// Library/Structures/AxesGroup/Acyclic/AxesGroupAcyclicAcrEntryRsp
{attribute 'pack_mode' := '1'} 
// ------------------------------------------------------------------------- 
//  SRCI Robot Library                                                
// ------------------------------------------------------------------------- 
//                                                                           
//  Object:      AxesGroupAcyclicAcrEntryRsp                                       
//  Author:      Thorsten Brach                                                
//  Date:        2024-06-01
//
//  Description:                                              
//   
//                                                                           
//  Copyright: 
//    (C) 2024 Thorsten Brach. All rights reserved                                                                                                                                            
//             Licensed under the LGPL-3.0 license.
//                                                                           
//  Disclaimer:                                                                           
//    This project is provided without any guarantee and can be used for   
//    private and commercial purposes. Any use is at the user’s 
//    own risk and responsibility.
//
// -------------------------------------------------------------------------
TYPE AxesGroupAcyclicAcrEntryRsp :
STRUCT
  /// Byte 00-03: Header
  Header : AxesGroupAcyclicAcrEntryRspHeader;
  /// Byte 04-07: Trigger sub header
  Trigger : AxesGroupAcyclicAcrEntryRspTrigger;
  /// Byte 08-xx: RSP Payload defined by type per CMD definition. Generated by Appl. Layer Task
  Payload : ARRAY[0..RobotLibraryParameter.TELEGRAM_PAYLOAD_MAX] OF BYTE;    
END_STRUCT
END_TYPE

// Library/Structures/AxesGroup/Acyclic/AxesGroupAcyclicAcrEntryRspBuffer
{attribute 'pack_mode' := '1'} 
// ------------------------------------------------------------------------- 
//  SRCI Robot Library                                                
// ------------------------------------------------------------------------- 
//                                                                           
//  Object:      AxesGroupAcyclicAcrEntryRspBuffer                                       
//  Author:      Thorsten Brach                                                
//  Date:        2024-06-01
//
//  Description:                                              
//   
//                                                                           
//  Copyright: 
//    (C) 2024 Thorsten Brach. All rights reserved                                                                                                                                            
//             Licensed under the LGPL-3.0 license.
//                                                                           
//  Disclaimer:                                                                           
//    This project is provided without any guarantee and can be used for   
//    private and commercial purposes. Any use is at the user’s 
//    own risk and responsibility.
//
// -------------------------------------------------------------------------
TYPE AxesGroupAcyclicAcrEntryRspBuffer :
STRUCT
  /// Timestamp
  Timestamp         : SystemTime;
  ///
  State             : BufferStateRsp;
  /// Payload defined by type per CMD definition. Processed by Appl. Layer Task.
  Payload           : ARRAY[0..RobotLibraryParameter.TELEGRAM_PAYLOAD_MAX] OF BYTE;
  /// Payload length
  PayloadLen        : UDINT;  
  /// Payload poiner   
  PayLoadPtr        : DWORD;
END_STRUCT
END_TYPE

// Library/Structures/AxesGroup/Acyclic/AxesGroupAcyclicAcrEntryRspHeader
{attribute 'pack_mode' := '1'} 
// ------------------------------------------------------------------------- 
//  SRCI Robot Library                                                
// ------------------------------------------------------------------------- 
//                                                                           
//  Object:      AxesGroupAcyclicAcrEntryRspHeader                                       
//  Author:      Thorsten Brach                                                
//  Date:        2024-06-01
//
//  Description:                                              
//   
//                                                                           
//  Copyright: 
//    (C) 2024 Thorsten Brach. All rights reserved                                                                                                                                            
//             Licensed under the LGPL-3.0 license.
//                                                                           
//  Disclaimer:                                                                           
//    This project is provided without any guarantee and can be used for   
//    private and commercial purposes. Any use is at the user’s 
//    own risk and responsibility.
//
// -------------------------------------------------------------------------
TYPE AxesGroupAcyclicAcrEntryRspHeader :
STRUCT
  /// Byte 00 : State  (Bit 0..3)
  State                : CmdMessageState; // ToDo : nicht sicher ob das richtig ist 
  /// Byte 00 : ParSeq (Bit 4..5)
  ParSeq               : BYTE;
  /// Byte 01 : Alarm Message Severity
  AlarmMessageSeverity : Severity;
  /// Byte 02 : Alarm Message Code
  AlarmMessageCode     : UINT;  
END_STRUCT
END_TYPE

// Library/Structures/AxesGroup/Acyclic/AxesGroupAcyclicAcrEntryRspTrigger
{attribute 'pack_mode' := '1'} 
// ------------------------------------------------------------------------- 
//  SRCI Robot Library                                                
// ------------------------------------------------------------------------- 
//                                                                           
//  Object:      AxesGroupAcyclicAcrEntryRspTrigger                                       
//  Author:      Thorsten Brach                                                
//  Date:        2024-06-01
//
//  Description:                                              
//   
//                                                                           
//  Copyright: 
//    (C) 2024 Thorsten Brach. All rights reserved                                                                                                                                            
//             Licensed under the LGPL-3.0 license.
//                                                                           
//  Disclaimer:                                                                           
//    This project is provided without any guarantee and can be used for   
//    private and commercial purposes. Any use is at the user’s 
//    own risk and responsibility.
//
// -------------------------------------------------------------------------
TYPE AxesGroupAcyclicAcrEntryRspTrigger :
STRUCT
  /// Number of Trigger based CMD invocations
  InvocationCounter       : USINT;
  /// Number of missed Triggers
  MissedInvocationCounter : USINT;
  /// FollowID of Trigger initiator
  OriginID                : WORD;
END_STRUCT
END_TYPE

// Library/Structures/AxesGroup/Acyclic/AxesGroupAcyclicExecutionOrderList
{attribute 'pack_mode' := '1'} 
// ------------------------------------------------------------------------- 
//  SRCI Robot Library                                                
// ------------------------------------------------------------------------- 
//                                                                           
//  Object:      AxesGroupAcyclicExecutionOrderList                                       
//  Author:      Thorsten Brach                                                
//  Date:        2024-06-01
//
//  Description:                                              
//   
//                                                                           
//  Copyright: 
//    (C) 2024 Thorsten Brach. All rights reserved                                                                                                                                            
//             Licensed under the LGPL-3.0 license.
//                                                                           
//  Disclaimer:                                                                           
//    This project is provided without any guarantee and can be used for   
//    private and commercial purposes. Any use is at the user’s 
//    own risk and responsibility.
//
// -------------------------------------------------------------------------
TYPE AxesGroupAcyclicExecutionOrderList :
STRUCT
  /// Command
  Command  : ARRAY [1..RobotLibraryParameter.ACTIVE_CMD_REGISTER_ENTRIES_MAX] OF UINT;
  /// Response
  Response : ARRAY [1..RobotLibraryParameter.ACTIVE_CMD_REGISTER_ENTRIES_MAX] OF UINT;
END_STRUCT
END_TYPE

// Library/Structures/AxesGroup/Cyclic/AxesGroupCyclic
{attribute 'pack_mode' := '1'} 
// ------------------------------------------------------------------------- 
//  SRCI Robot Library                                                
// ------------------------------------------------------------------------- 
//                                                                           
//  Object:      AxesGroupCyclic                                       
//  Author:      Thorsten Brach                                                
//  Date:        2024-06-01
//
//  Description:                                              
//   
//                                                                           
//  Copyright: 
//    (C) 2024 Thorsten Brach. All rights reserved                                                                                                                                            
//             Licensed under the LGPL-3.0 license.
//                                                                           
//  Disclaimer:                                                                           
//    This project is provided without any guarantee and can be used for   
//    private and commercial purposes. Any use is at the user’s 
//    own risk and responsibility.
//
// -------------------------------------------------------------------------
TYPE AxesGroupCyclic :
STRUCT
  /// Cyclic data from PLC to Robot 
  PlcToRob : AxesGroupCyclicPlcToRob;
  /// Cyclic data from Robot to PLC
  RobToPlc : AxesGroupCyclicRobToPlc;
END_STRUCT
END_TYPE

// Library/Structures/AxesGroup/Cyclic/AxesGroupCyclicPlcToRob
{attribute 'pack_mode' := '1'} 
// ------------------------------------------------------------------------- 
//  SRCI Robot Library                                                
// ------------------------------------------------------------------------- 
//                                                                           
//  Object:      AxesGroupCyclicPlcToRob                                       
//  Author:      Thorsten Brach                                                
//  Date:        2024-06-01
//
//  Description:                                              
//   
//                                                                           
//  Copyright: 
//    (C) 2024 Thorsten Brach. All rights reserved                                                                                                                                            
//             Licensed under the LGPL-3.0 license.
//                                                                           
//  Disclaimer:                                                                           
//    This project is provided without any guarantee and can be used for   
//    private and commercial purposes. Any use is at the user’s 
//    own risk and responsibility.
//
// -------------------------------------------------------------------------
TYPE AxesGroupCyclicPlcToRob :
STRUCT
  /// Version of SRCI specification
  /// Bit 0-4 : Minor version = Features        (0..31)
  /// Bit 5-7 : Major version = Breaking change (0..07)
  SRCIVersion            : VersionStruct;
  /// Fast stop trigger 
  FastStop               : BYTE;
  /// Connection alive signal
  LifeSign               : BYTE;
  /// Number of Bytes of the frame to be used for the telegram of the given Axisgroup. Direction client to server
  TelegramLengthPlcToRob : UINT;
  /// Number of Bytes of the frame to be used for the telegram of the given Axisgroup. Direction server to client
  TelegramLengthRobToPlc : UINT;
  /// Control AxesGroupID Telegtam state control
  AxesGroupID            : BYTE;
  /// Telegram state control
  Control                : ControlHalfByte;
  /// Reserved for later versions
  Reserved               : BYTE;
  /// Configuration of the optional cyclic data. Direction client to server
  TelegramNumberPlcToRob : UINT;
  /// Configuration of the optional cyclic data. Direction server to client
  TelegramNumberRobToPlc : UINT;
  /// Date of the client in the format days since 1990.01.01
  ClientDate             : IEC_DATE;
  /// Time in the clients time zone in the format milliseconds since start of day
  ClientTime             : IEC_TIME;    
  ///Index of tool of returned position
  /// •     -1: Currently used tool on RC
  /// •      0: Flange (default)
  /// • 1..254: Tool frames
  ToolNo                 : INT;
  /// Index of frame of returned position
  /// •     -1: Currently used frame on RC
  /// •      0: WCS (default)
  /// • 1..254: User frames
  FrameNo                : INT;
END_STRUCT
END_TYPE

// Library/Structures/AxesGroup/Cyclic/AxesGroupCyclicRobToPlc
{attribute 'pack_mode' := '1'} 
// ------------------------------------------------------------------------- 
//  SRCI Robot Library                                                
// ------------------------------------------------------------------------- 
//                                                                           
//  Object:      AxesGroupCyclicRobToPlc                                       
//  Author:      Thorsten Brach                                                
//  Date:        2024-06-01
//
//  Description:                                              
//   
//                                                                           
//  Copyright: 
//    (C) 2024 Thorsten Brach. All rights reserved                                                                                                                                            
//             Licensed under the LGPL-3.0 license.
//                                                                           
//  Disclaimer:                                                                           
//    This project is provided without any guarantee and can be used for   
//    private and commercial purposes. Any use is at the user’s 
//    own risk and responsibility.
//
// -------------------------------------------------------------------------
TYPE AxesGroupCyclicRobToPlc :
STRUCT
  /// Version of SRCI specification
  /// Bit 0-4 : Minor version = Features        (0..31)
  /// Bit 5-7 : Major version = Breaking change (0..07)
  SRCIVersion   : VersionStruct;
  /// Connection alive signal
  LifeSign      : BYTE;
  /// Reserved byte
  Reserved      : BYTE;
  /// Initialization and Telegram control state
  TelegramState : TelegramState;
  /// Combination of various RA related states.
  StatusRobotArm: RaStatusWord;
  /// Actual override in percentage encoding 
  Override      : UINT;  
END_STRUCT
END_TYPE

// Library/Structures/AxesGroup/CyclicOptional/Internal/AxesGroupCyclicOptionalDataCartesianPosition
{attribute 'pack_mode' := '1'} 
// ------------------------------------------------------------------------- 
//  SRCI Robot Library                                                
// ------------------------------------------------------------------------- 
//                                                                           
//  Object:      AxesGroupCyclicOptionalDataCartesianPosition                                       
//  Author:      Thorsten Brach                                                
//  Date:        2024-06-01
//
//  Description:                                              
//   
//                                                                           
//  Copyright: 
//    (C) 2024 Thorsten Brach. All rights reserved                                                                                                                                            
//             Licensed under the LGPL-3.0 license.
//                                                                           
//  Disclaimer:                                                                           
//    This project is provided without any guarantee and can be used for   
//    private and commercial purposes. Any use is at the user’s 
//    own risk and responsibility.
//
// -------------------------------------------------------------------------
TYPE AxesGroupCyclicOptionalDataCartesianPosition EXTENDS  RobotCartesianPositionShort :
STRUCT
  /// indicates that this optional parameter will be used
  Active           : BOOL;
  /// corresponding coordinate systems
  CoordinateSystem : RobotCoordinateSystemParameters; 
END_STRUCT
END_TYPE

// Library/Structures/AxesGroup/CyclicOptional/Internal/AxesGroupCyclicOptionalDataCartesianPositionExt
{attribute 'pack_mode' := '1'} 
// ------------------------------------------------------------------------- 
//  SRCI Robot Library                                                
// ------------------------------------------------------------------------- 
//                                                                           
//  Object:      AxesGroupCyclicOptionalDataCartesianPositionExt                                       
//  Author:      Thorsten Brach                                                
//  Date:        2024-06-01
//
//  Description:                                              
//   
//                                                                           
//  Copyright: 
//    (C) 2024 Thorsten Brach. All rights reserved                                                                                                                                            
//             Licensed under the LGPL-3.0 license.
//                                                                           
//  Disclaimer:                                                                           
//    This project is provided without any guarantee and can be used for   
//    private and commercial purposes. Any use is at the user’s 
//    own risk and responsibility.
//
// -------------------------------------------------------------------------
TYPE AxesGroupCyclicOptionalDataCartesianPositionExt EXTENDS RobotCartesianPositionExt :
STRUCT
  /// indicates that this optional parameter will be used
  Active : BOOL;
END_STRUCT
END_TYPE

// Library/Structures/AxesGroup/CyclicOptional/Internal/AxesGroupCyclicOptionalDataCurrent
{attribute 'pack_mode' := '1'} 
// ------------------------------------------------------------------------- 
//  SRCI Robot Library                                                
// ------------------------------------------------------------------------- 
//                                                                           
//  Object:      AxesGroupCyclicOptionalDataJointCurrent                                       
//  Author:      Thorsten Brach                                                
//  Date:        2024-06-01
//
//  Description:                                              
//   
//                                                                           
//  Copyright: 
//    (C) 2024 Thorsten Brach. All rights reserved                                                                                                                                            
//             Licensed under the LGPL-3.0 license.
//                                                                           
//  Disclaimer:                                                                           
//    This project is provided without any guarantee and can be used for   
//    private and commercial purposes. Any use is at the user’s 
//    own risk and responsibility.
//
// -------------------------------------------------------------------------
TYPE AxesGroupCyclicOptionalDataCurrent EXTENDS RobotJointCurrentShort :
STRUCT
    /// indicates that this optional parameter will be used
  Active : BOOL;
END_STRUCT
END_TYPE

// Library/Structures/AxesGroup/CyclicOptional/Internal/AxesGroupCyclicOptionalDataCurrentExt
{attribute 'pack_mode' := '1'} 
// ------------------------------------------------------------------------- 
//  SRCI Robot Library                                                
// ------------------------------------------------------------------------- 
//                                                                           
//  Object:      AxesGroupCyclicOptionalDataJointCurrentExt                                       
//  Author:      Thorsten Brach                                                
//  Date:        2024-06-01
//
//  Description:                                              
//   
//                                                                           
//  Copyright: 
//    (C) 2024 Thorsten Brach. All rights reserved                                                                                                                                            
//             Licensed under the LGPL-3.0 license.
//                                                                           
//  Disclaimer:                                                                           
//    This project is provided without any guarantee and can be used for   
//    private and commercial purposes. Any use is at the user’s 
//    own risk and responsibility.
//
// -------------------------------------------------------------------------
TYPE AxesGroupCyclicOptionalDataCurrentExt EXTENDS RobotJointCurrentExt :
STRUCT
    /// indicates that this optional parameter will be used
  Active : BOOL;
END_STRUCT
END_TYPE

// Library/Structures/AxesGroup/CyclicOptional/Internal/AxesGroupCyclicOptionalDataForce
{attribute 'pack_mode' := '1'} 
// ------------------------------------------------------------------------- 
//  SRCI Robot Library                                                
// ------------------------------------------------------------------------- 
//                                                                           
//  Object:      AxesGroupCyclicOptionalDataCartesianForce                                       
//  Author:      Thorsten Brach                                                
//  Date:        2024-06-01
//
//  Description:                                              
//   
//                                                                           
//  Copyright: 
//    (C) 2024 Thorsten Brach. All rights reserved                                                                                                                                            
//             Licensed under the LGPL-3.0 license.
//                                                                           
//  Disclaimer:                                                                           
//    This project is provided without any guarantee and can be used for   
//    private and commercial purposes. Any use is at the user’s 
//    own risk and responsibility.
//
// -------------------------------------------------------------------------
TYPE AxesGroupCyclicOptionalDataForce EXTENDS RobotCartesianForceShort:
STRUCT
  /// indicates that this optional parameter will be used
  Active           : BOOL;
END_STRUCT
END_TYPE

// Library/Structures/AxesGroup/CyclicOptional/Internal/AxesGroupCyclicOptionalDataForceExt
{attribute 'pack_mode' := '1'} 
// ------------------------------------------------------------------------- 
//  SRCI Robot Library                                                
// ------------------------------------------------------------------------- 
//                                                                           
//  Object:      AxesGroupCyclicOptionalDataCartesianForceExt                                       
//  Author:      Thorsten Brach                                                
//  Date:        2024-06-01
//
//  Description:                                              
//   
//                                                                           
//  Copyright: 
//    (C) 2024 Thorsten Brach. All rights reserved                                                                                                                                            
//             Licensed under the LGPL-3.0 license.
//                                                                           
//  Disclaimer:                                                                           
//    This project is provided without any guarantee and can be used for   
//    private and commercial purposes. Any use is at the user’s 
//    own risk and responsibility.
//
// -------------------------------------------------------------------------
TYPE AxesGroupCyclicOptionalDataForceExt EXTENDS RobotCartesianForceExt:
STRUCT
  /// indicates that this optional parameter will be used
  Active           : BOOL;
END_STRUCT
END_TYPE

// Library/Structures/AxesGroup/CyclicOptional/Internal/AxesGroupCyclicOptionalDataJointPosition
{attribute 'pack_mode' := '1'} 
// ------------------------------------------------------------------------- 
//  SRCI Robot Library                                                
// ------------------------------------------------------------------------- 
//                                                                           
//  Object:      AxesGroupCyclicOptionalDataJointPosition                                       
//  Author:      Thorsten Brach                                                
//  Date:        2024-06-01
//
//  Description:                                              
//   
//                                                                           
//  Copyright: 
//    (C) 2024 Thorsten Brach. All rights reserved                                                                                                                                            
//             Licensed under the LGPL-3.0 license.
//                                                                           
//  Disclaimer:                                                                           
//    This project is provided without any guarantee and can be used for   
//    private and commercial purposes. Any use is at the user’s 
//    own risk and responsibility.
//
// -------------------------------------------------------------------------
TYPE AxesGroupCyclicOptionalDataJointPosition EXTENDS RobotJointPositionShort :
STRUCT
    /// indicates that this optional parameter will be used
  Active : BOOL;
END_STRUCT
END_TYPE

// Library/Structures/AxesGroup/CyclicOptional/Internal/AxesGroupCyclicOptionalDataJointPositionExt
{attribute 'pack_mode' := '1'} 
// ------------------------------------------------------------------------- 
//  SRCI Robot Library                                                
// ------------------------------------------------------------------------- 
//                                                                           
//  Object:      AxesGroupCyclicOptionalDataJointPositionExt                                       
//  Author:      Thorsten Brach                                                
//  Date:        2024-06-01
//
//  Description:                                              
//   
//                                                                           
//  Copyright: 
//    (C) 2024 Thorsten Brach. All rights reserved                                                                                                                                            
//             Licensed under the LGPL-3.0 license.
//                                                                           
//  Disclaimer:                                                                           
//    This project is provided without any guarantee and can be used for   
//    private and commercial purposes. Any use is at the user’s 
//    own risk and responsibility.
//
// -------------------------------------------------------------------------
TYPE AxesGroupCyclicOptionalDataJointPositionExt EXTENDS RobotJointPositionExt :
STRUCT
    /// indicates that this optional parameter will be used
  Active : BOOL;
END_STRUCT
END_TYPE

// Library/Structures/AxesGroup/CyclicOptional/Internal/AxesGroupCyclicOptionalDataSubProgram
{attribute 'pack_mode' := '1'} 
// ------------------------------------------------------------------------- 
//  SRCI Robot Library                                                
// ------------------------------------------------------------------------- 
//                                                                           
//  Object:      AxesGroupCyclicOptionalDataSubProgram                                       
//  Author:      Thorsten Brach                                                
//  Date:        2024-06-01
//
//  Description:                                              
//   
//                                                                           
//  Copyright: 
//    (C) 2024 Thorsten Brach. All rights reserved                                                                                                                                            
//             Licensed under the LGPL-3.0 license.
//                                                                           
//  Disclaimer:                                                                           
//    This project is provided without any guarantee and can be used for   
//    private and commercial purposes. Any use is at the user’s 
//    own risk and responsibility.
//
// -------------------------------------------------------------------------
TYPE AxesGroupCyclicOptionalDataSubProgram EXTENDS RobotSubProgramData :
STRUCT
  /// indicates that this optional parameter will be used
  Active : BOOL;
END_STRUCT
END_TYPE

// Library/Structures/AxesGroup/CyclicOptional/AxesGroupCyclicOptionalData
{attribute 'pack_mode' := '1'} 
// ------------------------------------------------------------------------- 
//  SRCI Robot Library                                                
// ------------------------------------------------------------------------- 
//                                                                           
//  Object:      AxesGroupCyclicOptionalData                                       
//  Author:      Thorsten Brach                                                
//  Date:        2024-06-01
//
//  Description:                                              
//   
//                                                                           
//  Copyright: 
//    (C) 2024 Thorsten Brach. All rights reserved                                                                                                                                            
//             Licensed under the LGPL-3.0 license.
//                                                                           
//  Disclaimer:                                                                           
//    This project is provided without any guarantee and can be used for   
//    private and commercial purposes. Any use is at the user’s 
//    own risk and responsibility.
//
// -------------------------------------------------------------------------
TYPE AxesGroupCyclicOptionalData :
STRUCT
  /// Optional cyclic data from PLC to Robot
  PlcToRob : AxesGroupCyclicOptionalDataPlcToRob;
  /// Optional cyclic data from Robot to PLC
  RobToPlc : AxesGroupCyclicOptionalDataRobToPlc;
END_STRUCT
END_TYPE

// Library/Structures/AxesGroup/CyclicOptional/AxesGroupCyclicOptionalDataPlcToRob
{attribute 'pack_mode' := '1'} 
// ------------------------------------------------------------------------- 
//  SRCI Robot Library                                                
// ------------------------------------------------------------------------- 
//                                                                           
//  Object:      vAxesGroupCyclicOptionalDataPlcToRob                                       
//  Author:      Thorsten Brach                                                
//  Date:        2024-06-01
//
//  Description:                                              
//   
//                                                                           
//  Copyright: 
//    (C) 2024 Thorsten Brach. All rights reserved                                                                                                                                            
//             Licensed under the LGPL-3.0 license.
//                                                                           
//  Disclaimer:                                                                           
//    This project is provided without any guarantee and can be used for   
//    private and commercial purposes. Any use is at the user’s 
//    own risk and responsibility.
//
// -------------------------------------------------------------------------
TYPE AxesGroupCyclicOptionalDataPlcToRob :
STRUCT
  /// Transmit cyclic data from PLC to RC for the usage in a subprogram on the RC called via the function “CallSubprogram”
  SubProgramData        :  AxesGroupCyclicOptionalDataSubProgram;
  /// short cartesian position with TCP position (X, Y,Z), rotation (RX, RY, RZ), configuration bytes (Config, TurnNumber), position of first external axis (E1) and corresponding coordinate systems (ToolNo, FrameNo)
  CartesianPosition     :  AxesGroupCyclicOptionalDataCartesianPosition;
  /// the external axis values for an extended cartesian position (E2, E3, E4, E5, E6) 
  /// When selected, Tool and Frame will automatically cyclically be sent from client to server.
  CartesianPositionExt  :  AxesGroupCyclicOptionalDataCartesianPositionExt;
  /// short axes position with joint values (J1, J2, J3,J4, J5, J6) and position of first external axis (E1)
  JointPosition         :  AxesGroupCyclicOptionalDataJointPosition;
  /// the external axis values for an extended joint position (E2, E3, E4, E5, E6)
  JointPositionExt      :  AxesGroupCyclicOptionalDataJointPositionExt;
  /// force with the divided forces in the individual directions (X, Y, Z, RX, RY, RZ)
  Force                 :  AxesGroupCyclicOptionalDataForce;
  /// current force for the external axis (E1, E2, E3, E4, E5, E6)
  ForceExt              :  AxesGroupCyclicOptionalDataForceExt;
END_STRUCT
END_TYPE

// Library/Structures/AxesGroup/CyclicOptional/AxesGroupCyclicOptionalDataRobToPlc
{attribute 'pack_mode' := '1'} 
// ------------------------------------------------------------------------- 
//  SRCI Robot Library                                                
// ------------------------------------------------------------------------- 
//                                                                           
//  Object:      AxesGroupCyclicOptionalDataRobToPlc                                       
//  Author:      Thorsten Brach                                                
//  Date:        2024-06-01
//
//  Description:                                              
//   
//                                                                           
//  Copyright: 
//    (C) 2024 Thorsten Brach. All rights reserved                                                                                                                                            
//             Licensed under the LGPL-3.0 license.
//                                                                           
//  Disclaimer:                                                                           
//    This project is provided without any guarantee and can be used for   
//    private and commercial purposes. Any use is at the user’s 
//    own risk and responsibility.
//
// -------------------------------------------------------------------------
TYPE AxesGroupCyclicOptionalDataRobToPlc :
STRUCT
  /// Transmit cyclic data from PLC to RC for the usage in a subprogram on the RC called via the function “CallSubprogram”
  SubProgramData        :  AxesGroupCyclicOptionalDataSubProgram;
  /// short cartesian position with TCP position (X, Y,Z), rotation (RX, RY, RZ), configuration bytes (Config, TurnNumber), position of first external axis (E1) and corresponding coordinate systems (ToolNo, FrameNo)
  CartesianPosition     :  AxesGroupCyclicOptionalDataCartesianPosition;
  /// the external axis values for an extended cartesian position (E2, E3, E4, E5, E6) 
  /// When selected, Tool and Frame will automatically cyclically be sent from client to server.
  CartesianPositionExt  :  AxesGroupCyclicOptionalDataCartesianPositionExt;
  /// short axes position with joint values (J1, J2, J3,J4, J5, J6) and position of first external axis (E1)
  JointPosition         :  AxesGroupCyclicOptionalDataJointPosition;
  /// the external axis values for an extended joint position (E2, E3, E4, E5, E6)
  JointPositionExt      :  AxesGroupCyclicOptionalDataJointPositionExt;
  /// force with the divided forces in the individual directions (X, Y, Z, RX, RY, RZ)
  Force                 :  AxesGroupCyclicOptionalDataForce;
  /// current force for the external axis (E1, E2, E3, E4, E5, E6)
  ForceExt              :  AxesGroupCyclicOptionalDataForceExt;
  /// ctual axes current of individual axes (J1, J2, J3, J4, J5, J6)
  Current               :  AxesGroupCyclicOptionalDataCurrent;
  /// actual current for the external axis (E1, E2,E3, E4, E5, E6)
  CurrentExt            :  AxesGroupCyclicOptionalDataCurrentExt;  
END_STRUCT
END_TYPE

// Library/Structures/AxesGroup/InternalData/AxesGroupInternalData
{attribute 'pack_mode' := '1'} 
// ------------------------------------------------------------------------- 
//  SRCI Robot Library                                                
// ------------------------------------------------------------------------- 
//                                                                           
//  Object:      AxesGroup                                       
//  Author:      Thorsten Brach                                                
//  Date:        2024-08-28
//
//  Description:                                              
//   
//                                                                           
//  Copyright: 
//    (C) 2024 Thorsten Brach. All rights reserved                                                                                                                                            
//             Licensed under the LGPL-3.0 license.
//                                                                           
//  Disclaimer:                                                                           
//    This project is provided without any guarantee and can be used for   
//    private and commercial purposes. Any use is at the user’s 
//    own risk and responsibility.
//
// -------------------------------------------------------------------------
TYPE AxesGroupInternalData :
STRUCT
  /// Current System Time
  SystemTime           : SystemTime;
    /// • TRUE: Function is supported by RC • FALSE: Function is not supported by RC See Table 6-14 for bit assignment.
  RCSupportedFunctions : RCSupportedFunctions;
  /// Online Change detected
  OnlineChange         : BOOL;  
  /// Rising edge for Online Change detected
  OnlineChange_R       : R_TRIG;  
  /// Falling edge for Online Change detected
  OnlineChange_F       : F_TRIG;  
  /// GroupReset active
  GroupReset           : BOOL; 
  /// Rising edge for GroupReset
  GroupReset_R         : R_TRIG;  
  /// Falling edge for GroupReset
  GroupReset_F         : F_TRIG;
  /// Counter of sequences to send
  SequenceCountSend    : DINT;
  /// Counter of sequences received
  SequenceCountRecv    : DINT;
  /// Counter of fragments to send
  FragmentCountSend    : ARRAY[0..1] OF DINT;
  /// Counter of fragments received
  FragmentCountRecv    : ARRAY[0..1] OF DINT;
  /// Current Sequence ID
  CurrentSEQ           : ARRAY[0..1] OF UINT;
  /// Current acknowledge ID
  CurrentACK           : ARRAY[0..1] OF UINT;  
  /// Current Sequence ID has changed -> send new data 
  NewSEQ               : ARRAY[0..1] OF BOOL;
  /// Last received acknowledge ID
  LastACK              : ARRAY[0..1] OF UINT;  
END_STRUCT
END_TYPE

// Library/Structures/AxesGroup/MessageLog/AxesGroupMessageLog
{attribute 'pack_mode' := '1'} 
// ------------------------------------------------------------------------- 
//  SRCI Robot Library                                                
// ------------------------------------------------------------------------- 
//                                                                           
//  Object:      AxesGroupMessageLog                                       
//  Author:      Thorsten Brach                                                
//  Date:        2024-06-01
//
//  Description:                                              
//   
//                                                                           
//  Copyright: 
//    (C) 2024 Thorsten Brach. All rights reserved                                                                                                                                            
//             Licensed under the LGPL-3.0 license.
//                                                                           
//  Disclaimer:                                                                           
//    This project is provided without any guarantee and can be used for   
//    private and commercial purposes. Any use is at the user’s 
//    own risk and responsibility.
//
// -------------------------------------------------------------------------
TYPE AxesGroupMessageLog :
STRUCT
  /// Amount of system log entries
  SystemLogEntries : UINT := DINT_TO_UINT(RobotLibraryParameter.SYSTEM_LOG_MAX);
  /// Amount of message log entries
  MessagesEntries  : UINT := DINT_TO_UINT(RobotLibraryParameter.MESSAGE_LOG_MAX);
  /// Logging level
  LogLevel         : LogLevel;
  /// System log
  SystemLog        : ARRAY[0..RobotLibraryParameter.SYSTEM_LOG_MAX] OF STRING(255);
  /// Message Log
  Messages         : ARRAY[0..RobotLibraryParameter.MESSAGE_LOG_MAX] OF AlarmMessage;
  /// Interface to an external logger
  ExternalLogger   : IMessageLogger;
END_STRUCT
END_TYPE

// Library/Structures/AxesGroup/Parameter/Cmd/AxesGroupParameterCmdEntry
{attribute 'pack_mode' := '1'} 
// ------------------------------------------------------------------------- 
//  SRCI Robot Library                                                
// ------------------------------------------------------------------------- 
//                                                                           
//  Object:      AxesGroupParameterCmdEntry                                       
//  Author:      Thorsten Brach                                                
//  Date:        2024-06-01
//
//  Description:                                              
//   
//                                                                           
//  Copyright: 
//    (C) 2024 Thorsten Brach. All rights reserved                                                                                                                                            
//             Licensed under the LGPL-3.0 license.
//                                                                           
//  Disclaimer:                                                                           
//    This project is provided without any guarantee and can be used for   
//    private and commercial purposes. Any use is at the user’s 
//    own risk and responsibility.
//
// -------------------------------------------------------------------------
TYPE AxesGroupParameterCmdEntry :
STRUCT
  /// User defined command name
  Name                 : STRING(20);
  ///
  CmdType              : CmdType; 
  ///
  Prio                 : PriorityLevel;
  ///
  HighPrio             : USINT;
  ///
  ExecMode             : ExecutionMode;
  ///
  SequenceFlag         : SequenceFlag;
  /// ID of Action that will be executed when this command is active
  /// • >0: Start Action - Start executing the Action function with the identical ListenerID.
  /// • <0: Stop Action  -  Stop executing the Action function with the identical ListenerID.
  /// • 0: No trigger (default)-  If no EmitterID is defined, the function will not trigger any Action during its execution
  /// For more information see section Triggers of this chapter or chapter 5.5.12.4.
  EmitterID            : ARRAY [0..3] OF SINT;
  /// ID of associated trigger function:
  /// • 0: No Trigger (default): No trigger related behavior
  /// • >0: Trigger:  Start executing, when the trigger function with the identical EmitterID is triggered.
  /// Always positive.
  /// For more information, see chapter 5.5.12 Triggers
  ListenerID           : SINT;
  ///
  ExecutionModeAllowed : ProcessingModeAllowed;
  ///
  LogParameter         : LogParameter;
  ///
  FunctionMode         : USINT; // ToDo ?
  ///
  CheckEmitterID       : SINT;
  ///
  CheckListenerID      : SINT;
END_STRUCT
END_TYPE

// Library/Structures/AxesGroup/Parameter/OptionalCyclic/AxesGroupParameterOptionalCyclic
{attribute 'pack_mode' := '1'} 
// ------------------------------------------------------------------------- 
//  SRCI Robot Library                                                
// ------------------------------------------------------------------------- 
//                                                                           
//  Object:      AxesGroupParameterOptionalCyclic                                       
//  Author:      Thorsten Brach                                                
//  Date:        2024-06-01
//
//  Description:                                              
//   
//                                                                           
//  Copyright: 
//    (C) 2024 Thorsten Brach. All rights reserved                                                                                                                                            
//             Licensed under the LGPL-3.0 license.
//                                                                           
//  Disclaimer:                                                                           
//    This project is provided without any guarantee and can be used for   
//    private and commercial purposes. Any use is at the user’s 
//    own risk and responsibility.
//
// -------------------------------------------------------------------------
TYPE AxesGroupParameterOptionalCyclic :
STRUCT
  /// Configuration of optional cyclic data send to the Robot
  PlcToRob : AxesGroupParameterOptionalCyclicPlcToRob;
  /// Configuration of optional cyclic data received from the Robot
  RobToPlc : AxesGroupParameterOptionalCyclicRobToPlc;
END_STRUCT
END_TYPE

// Library/Structures/AxesGroup/Parameter/OptionalCyclic/AxesGroupParameterOptionalCyclicPlcToRob
{attribute 'pack_mode' := '1'} 
// ------------------------------------------------------------------------- 
//  SRCI Robot Library                                                
// ------------------------------------------------------------------------- 
//                                                                           
//  Object:      AxesGroupParameterOptionalCyclicPlcToRob                                       
//  Author:      Thorsten Brach                                                
//  Date:        2024-06-01
//
//  Description:                                              
//   
//                                                                           
//  Copyright: 
//    (C) 2024 Thorsten Brach. All rights reserved                                                                                                                                            
//             Licensed under the LGPL-3.0 license.
//                                                                           
//  Disclaimer:                                                                           
//    This project is provided without any guarantee and can be used for   
//    private and commercial purposes. Any use is at the user’s 
//    own risk and responsibility.
//
// -------------------------------------------------------------------------
TYPE AxesGroupParameterOptionalCyclicPlcToRob :
STRUCT
  /// Bit 00: 
  /// Transmit cyclic data from PLC to RC for the usage in a subprogram on the RC called via the function “CallSubprogram”
  UseCallSubprogram       : BOOL;
  /// Bit 01: 
  /// Send a short cartesian position with TCP position (X, Y,Z), rotation (RX, RY, RZ), 
  /// configuration bytes (Config, TurnNumber), position of first external axis (E1) and corresponding coordinate systems (ToolNo, FrameNo)
  UseCartesianPosition    : BOOL;
  /// Bit 02: 
  /// Send a short axes position with joint values (J1, J2, J3, J4, J5, J6) and position of first external axis (E1)
  UseJointPosition        : BOOL;
  /// Bit 03: 
  /// Send the force with the divided forces in the individual directions (X, Y, Z, RX, RY, RZ)
  UseForce                : BOOL;
  /// Bit 04:
  Bit04                   : BOOL;
  /// Bit 05:
  Bit05                   : BOOL;
  /// Bit 06:
  Bit06                   : BOOL;
  /// Bit 07:
  Bit07                   : BOOL;  
  /// Bit 08: 
  /// Set to 1 to define two Sequences in one Telegram. 
  /// If activated, 2 sequences also has to be activated in the ServerClient direction
  UseTwoSequences         : BOOL;
  /// Bit 09: 
  /// Send the external axis values for an extended cartesian position (E2, E3, E4, E5, E6)
  UseCartesianPositionExt : BOOL;
  /// Bit 10: 
  /// Send the external axis values for an extended joint position (E2, E3, E4, E5, E6)
  UseJointPositionExt     : BOOL;
  /// Bit 11:
  Bit11                   : BOOL;
  /// Bit 12:
  Bit12                   : BOOL;
  /// Bit 13:
  Bit13                   : BOOL;
  /// Bit 14:
  Bit14                   : BOOL;
  /// Bit 15:
  Bit15                   : BOOL;  
END_STRUCT
END_TYPE

// Library/Structures/AxesGroup/Parameter/OptionalCyclic/AxesGroupParameterOptionalCyclicRobToPlc
{attribute 'pack_mode' := '1'} 
// ------------------------------------------------------------------------- 
//  SRCI Robot Library                                                
// ------------------------------------------------------------------------- 
//                                                                           
//  Object:      AxesGroupParameterOptionalCyclicRobToPlc                                       
//  Author:      Thorsten Brach                                                
//  Date:        2024-06-01
//
//  Description:                                              
//   
//                                                                           
//  Copyright: 
//    (C) 2024 Thorsten Brach. All rights reserved                                                                                                                                            
//             Licensed under the LGPL-3.0 license.
//                                                                           
//  Disclaimer:                                                                           
//    This project is provided without any guarantee and can be used for   
//    private and commercial purposes. Any use is at the user’s 
//    own risk and responsibility.
//
// -------------------------------------------------------------------------
TYPE AxesGroupParameterOptionalCyclicRobToPlc :
STRUCT
  /// Bit 00: 
  /// Transmit cyclic data from PLC to RC for the usage in a subprogram on the RC called via the function “CallSubprogram”
  UseCallSubprogram       : BOOL;
  /// Bit 01: 
  /// Send a short cartesian position with TCP position (X, Y,Z), rotation (RX, RY, RZ), 
  /// configuration bytes (Config, TurnNumber), position of first external axis (E1) and corresponding coordinate systems (ToolNo, FrameNo)
  UseCartesianPosition    : BOOL;
  /// Bit 02: 
  /// Send a short axes position with joint values (J1, J2, J3, J4, J5, J6) and position of first external axis (E1)
  UseJointPosition        : BOOL;
  /// Bit 03: 
  /// Send the force with the divided forces in the individual directions (X, Y, Z, RX, RY, RZ)
  UseForce                : BOOL;
  /// Bit 04:
  /// Transmit actual axes current of individual axes (J1, J2, J3, J4, J5, J6)
  UseCurrent              : BOOL;
  /// Bit 05:
  Bit05                   : BOOL;
  /// Bit 06:
  Bit06                   : BOOL;
  /// Bit 07:
  Bit07                   : BOOL;  
  /// Bit 08: 
  /// Set to 1 to define two Sequences in one Telegram. 
  /// If activated, 2 sequences also has to be activated in the ServerClient direction
  UseTwoSequences         : BOOL;
  /// Bit 09: 
  /// Send the external axis values for an extended cartesian position (E2, E3, E4, E5, E6)
  UseCartesianPositionExt : BOOL;
  /// Bit 10: 
  /// Send the external axis values for an extended joint position (E2, E3, E4, E5, E6)
  UseJointPositionExt     : BOOL;
  /// Bit 11:
  /// Transmit the current force for the external axis (E1, E2, E3, E4, E5, E6)
  UseForceExt             : BOOL;
  /// Bit 12:
  /// Transmit the actual current for the external axis (E1, E2, E3, E4, E5, E6)
  UseCurrentExt           : BOOL;
  /// Bit 13:
  Bit13                   : BOOL;
  /// Bit 14:
  Bit14                   : BOOL;
  /// Bit 15:
  Bit15                   : BOOL;  
END_STRUCT
END_TYPE

// Library/Structures/AxesGroup/Parameter/Plc/AxesGroupParameterPlc
{attribute 'pack_mode' := '1'} 
// ------------------------------------------------------------------------- 
//  SRCI Robot Library                                                
// ------------------------------------------------------------------------- 
//                                                                           
//  Object:      AxesGroupParameterPlc                                       
//  Author:      Thorsten Brach                                                
//  Date:        2024-06-01
//
//  Description:                                              
//   
//                                                                           
//  Copyright: 
//    (C) 2024 Thorsten Brach. All rights reserved                                                                                                                                            
//             Licensed under the LGPL-3.0 license.
//                                                                           
//  Disclaimer:                                                                           
//    This project is provided without any guarantee and can be used for   
//    private and commercial purposes. Any use is at the user’s 
//    own risk and responsibility.
//
// -------------------------------------------------------------------------
TYPE AxesGroupParameterPlc :
STRUCT
  (*
  /// Manufactured ID
  ManufacturedID       : UINT;
  /// Order ID
  OrderID              : STRING(20);
  /// Serial Number
  SerialNumber         : STRING(16);
  /// Firmware Version
  FirmwareVersion      : STRING(8);
  /// Client Interface Version
  InterfaceVersion     : STRING(8);
  /// Synchronization Modes
  SynchronizationModes : SynchronizationModes;  
*)
  Parameter            : AxesGroupParameterPlcParameter;  
  OptionalCyclic       : AxesGroupParameterPlcOptionalCyclic;
END_STRUCT
END_TYPE

// Library/Structures/AxesGroup/Parameter/Plc/AxesGroupParameterPlcOptionalCyclic
{attribute 'pack_mode' := '1'} 
// ------------------------------------------------------------------------- 
//  SRCI Robot Library                                                
// ------------------------------------------------------------------------- 
//                                                                           
//  Object:      AxesGroupParameterPlcOptionalCyclic                                       
//  Author:      Thorsten Brach                                                
//  Date:        2024-11-30
//
//  Description:                                              
//   
//                                                                           
//  Copyright: 
//    (C) 2024 Thorsten Brach. All rights reserved                                                                                                                                            
//             Licensed under the LGPL-3.0 license.
//                                                                           
//  Disclaimer:                                                                           
//    This project is provided without any guarantee and can be used for   
//    private and commercial purposes. Any use is at the user’s 
//    own risk and responsibility.
//
// -------------------------------------------------------------------------
TYPE AxesGroupParameterPlcOptionalCyclic :
STRUCT
  /// Bit 00: 
  /// Transmit cyclic data from PLC to RC for the usage in a subprogram on the RC called via the function “CallSubprogram”
  UseCallSubprogram       : BOOL;
  /// Bit 01: 
  /// Send a short cartesian position with TCP position (X, Y,Z), rotation (RX, RY, RZ), 
  /// configuration bytes (Config, TurnNumber), position of first external axis (E1) and corresponding coordinate systems (ToolNo, FrameNo)
  UseCartesianPosition    : BOOL;
  /// Bit 02: 
  /// Send a short axes position with joint values (J1, J2, J3, J4, J5, J6) and position of first external axis (E1)
  UseJointPosition        : BOOL;
  /// Bit 03: 
  /// Send the force with the divided forces in the individual directions (X, Y, Z, RX, RY, RZ)
  UseForce                : BOOL;
  /// Bit 04:
  Bit04                   : BOOL;
  /// Bit 05:
  Bit05                   : BOOL;
  /// Bit 06:
  Bit06                   : BOOL;
  /// Bit 07:
  Bit07                   : BOOL;  
  /// Bit 08: 
  /// Set to 1 to define two Sequences in one Telegram. 
  /// If activated, 2 sequences also has to be activated in the ServerClient direction
  UseTwoSequences         : BOOL;
  /// Bit 09: 
  /// Send the external axis values for an extended cartesian position (E2, E3, E4, E5, E6)
  UseCartesianPositionExt : BOOL;
  /// Bit 10: 
  /// Send the external axis values for an extended joint position (E2, E3, E4, E5, E6)
  UseJointPositionExt     : BOOL;
  /// Bit 11:
  Bit11                   : BOOL;
  /// Bit 12:
  Bit12                   : BOOL;
  /// Bit 13:
  Bit13                   : BOOL;
  /// Bit 14:
  Bit14                   : BOOL;
  /// Bit 15:
  Bit15                   : BOOL;  
END_STRUCT
END_TYPE

// Library/Structures/AxesGroup/Parameter/Plc/AxesGroupParameterPlcParameter
{attribute 'pack_mode' := '1'} 
// ------------------------------------------------------------------------- 
//  SRCI Robot Library                                                
// ------------------------------------------------------------------------- 
//                                                                           
//  Object:      AxesGroupParameterPlcParameter                                       
//  Author:      Thorsten Brach                                                
//  Date:        2024-11-30
//
//  Description:                                              
//   
//                                                                           
//  Copyright: 
//    (C) 2024 Thorsten Brach. All rights reserved                                                                                                                                            
//             Licensed under the LGPL-3.0 license.
//                                                                           
//  Disclaimer:                                                                           
//    This project is provided without any guarantee and can be used for   
//    private and commercial purposes. Any use is at the user’s 
//    own risk and responsibility.
//
// -------------------------------------------------------------------------
TYPE AxesGroupParameterPlcParameter :
STRUCT
  /// Manufactured ID
  ManufacturedID       : UINT;
  /// Order ID
  OrderID              : STRING(20);
  /// Serial Number
  SerialNumber         : STRING(16);
  /// Firmware Version
  FirmwareVersion      : STRING(8);
  /// Client Interface Version
  InterfaceVersion     : STRING(8);
  /// Synchronization Modes
  SynchronizationModes : SynchronizationModes;  
  /// Optional Cyclic values
  OptionalCyclic       : AxesGroupParameterPlcOptionalCyclic;
END_STRUCT               
END_TYPE

// Library/Structures/AxesGroup/Parameter/Rob/AxesGroupParameterRob
{attribute 'pack_mode' := '1'} 
// ------------------------------------------------------------------------- 
//  SRCI Robot Library                                                
// ------------------------------------------------------------------------- 
//                                                                           
//  Object:      AxesGroupParameterRob                                       
//  Author:      Thorsten Brach                                                
//  Date:        2024-06-01
//
//  Description:                                              
//   
//                                                                           
//  Copyright: 
//    (C) 2024 Thorsten Brach. All rights reserved                                                                                                                                            
//             Licensed under the LGPL-3.0 license.
//                                                                           
//  Disclaimer:                                                                           
//    This project is provided without any guarantee and can be used for   
//    private and commercial purposes. Any use is at the user’s 
//    own risk and responsibility.
//
// -------------------------------------------------------------------------
TYPE AxesGroupParameterRob :
STRUCT  
  (*
  /// User defined robot name
  RobotName                 : STRING(20);
  /// Returns a metric of how many CMDs it can receive and manage at the same time
  LengthACR                 : UINT;
  /// Highest index of available tools on the RC.
  HighestToolIndex          : USINT;
  /// Highest index of available frames on the RC.
  HighestFrameIndex         : USINT;
  /// Highest index of available loads on the RC.
  HighestLoadIndex          : USINT;
  /// Highest index of available work areas on the RC.
  HighestWorkAreaIndex      : USINT;
  /// Datas which are synchronized
  DataInSync                : DataInSync;
  /// Index of tool changed on RC
  ChangeIndexTool           : USINT;
  /// Index of frame changed on RC
  ChangeIndexFrame          : USINT;
  /// Index of load changed on RC
  ChangeIndexLoad           : USINT;
  ///Index of work area changed on RC
  ChangeIndexWorkArea       : USINT;
  /// Working hours of an RA connected to the RC
  RAWorkingHours            : UDINT;
  /// Signals that a brake test is required in the defined monitoring time (see chapter 6.5.27)
  BrakeTestRequired         : BOOL;
  /// StepMode is active and set to ExactStop (see chapter 6.1.3)
  StepModeExactStopActive   : BOOL;
  /// StepMode is active and set to Blending (see chapter 6.1.3)
  StepModeBlendingActive    : BOOL;
  /// PathAccuracyMode is active (see chapter 6.5.22)
  PathAccuracyMode          : BOOL;
  /// AvoidSingularity is active (see chapter 6.5.23)
  AvoidSingularity          : BOOL;
  /// CollisionDetection is active (see chapter 6.5.35)
  CollisionDetectionEnabled : BOOL;
  /// Cyclic dynamics status bit Accelerating is supported by RC (see chapter 5.5.3.2)
  AcceleratingSupported     : BOOL;
  /// Cyclic dynamics status bit Decelerating is supported by RC (see chapter 5.5.3.2)
  DecceleratingSupported    : BOOL;
  /// Cyclic dynamics status bit ConstantVelocity is supported by RC (see chapter 5.5.3.2)
  ConstantVelocitySupported : BOOL;
  /// Total system hours of an RA connected to the RC. Must not be modifiable by the user.
  /// •  0: Invalid
  /// • >1: Total system hours
  RCWorkingHours            : UDINT;
*)  
  /// 
  Parameter                 : AxesGroupParameterRobParameter;
  /// 
  OptionalCyclic            : AxesGroupParameterRobOptionalCyclic;
END_STRUCT
END_TYPE

// Library/Structures/AxesGroup/Parameter/Rob/AxesGroupParameterRobOptionalCyclic
{attribute 'pack_mode' := '1'} 
// ------------------------------------------------------------------------- 
//  SRCI Robot Library                                                
// ------------------------------------------------------------------------- 
//                                                                           
//  Object:      AxesGroupParameterOptionalCyclicRobToPlc                                       
//  Author:      Thorsten Brach                                                
//  Date:        2024-06-01
//
//  Description:                                              
//   
//                                                                           
//  Copyright: 
//    (C) 2024 Thorsten Brach. All rights reserved                                                                                                                                            
//             Licensed under the LGPL-3.0 license.
//                                                                           
//  Disclaimer:                                                                           
//    This project is provided without any guarantee and can be used for   
//    private and commercial purposes. Any use is at the user’s 
//    own risk and responsibility.
//
// -------------------------------------------------------------------------
TYPE AxesGroupParameterRobOptionalCyclic :
STRUCT
  /// Bit 00: 
  /// Transmit cyclic data from PLC to RC for the usage in a subprogram on the RC called via the function “CallSubprogram”
  UseCallSubprogram       : BOOL;
  /// Bit 01: 
  /// Send a short cartesian position with TCP position (X, Y,Z), rotation (RX, RY, RZ), 
  /// configuration bytes (Config, TurnNumber), position of first external axis (E1) and corresponding coordinate systems (ToolNo, FrameNo)
  UseCartesianPosition    : BOOL;
  /// Bit 02: 
  /// Send a short axes position with joint values (J1, J2, J3, J4, J5, J6) and position of first external axis (E1)
  UseJointPosition        : BOOL;
  /// Bit 03: 
  /// Send the force with the divided forces in the individual directions (X, Y, Z, RX, RY, RZ)
  UseForce                : BOOL;
  /// Bit 04:
  /// Transmit actual axes current of individual axes (J1, J2, J3, J4, J5, J6)
  UseCurrent              : BOOL;
  /// Bit 05:
  Bit05                   : BOOL;
  /// Bit 06:
  Bit06                   : BOOL;
  /// Bit 07:
  Bit07                   : BOOL;  
  /// Bit 08: 
  /// Set to 1 to define two Sequences in one Telegram. 
  /// If activated, 2 sequences also has to be activated in the ServerClient direction
  UseTwoSequences         : BOOL;
  /// Bit 09: 
  /// Send the external axis values for an extended cartesian position (E2, E3, E4, E5, E6)
  UseCartesianPositionExt : BOOL;
  /// Bit 10: 
  /// Send the external axis values for an extended joint position (E2, E3, E4, E5, E6)
  UseJointPositionExt     : BOOL;
  /// Bit 11:
  /// Transmit the current force for the external axis (E1, E2, E3, E4, E5, E6)
  UseForceExt             : BOOL;
  /// Bit 12:
  /// Transmit the actual current for the external axis (E1, E2, E3, E4, E5, E6)
  UseCurrentExt           : BOOL;
  /// Bit 13:
  Bit13                   : BOOL;
  /// Bit 14:
  Bit14                   : BOOL;
  /// Bit 15:
  Bit15                   : BOOL;  
END_STRUCT
END_TYPE

// Library/Structures/AxesGroup/Parameter/Rob/AxesGroupParameterRobParameter
{attribute 'pack_mode' := '1'} 
// ------------------------------------------------------------------------- 
//  SRCI Robot Library                                                
// ------------------------------------------------------------------------- 
//                                                                           
//  Object:      AxesGroupParameterRob                                       
//  Author:      Thorsten Brach                                                
//  Date:        2024-06-01
//
//  Description:                                              
//   
//                                                                           
//  Copyright: 
//    (C) 2024 Thorsten Brach. All rights reserved                                                                                                                                            
//             Licensed under the LGPL-3.0 license.
//                                                                           
//  Disclaimer:                                                                           
//    This project is provided without any guarantee and can be used for   
//    private and commercial purposes. Any use is at the user’s 
//    own risk and responsibility.
//
// -------------------------------------------------------------------------
TYPE AxesGroupParameterRobParameter :
STRUCT  
  /// User defined robot name
  RobotName                 : STRING(20);
  /// Returns a metric of how many CMDs it can receive and manage at the same time
  /// must be initialized with a value > 3, because during the interface initialization at least 3 commands are executed
  /// after ReadRobotData command the value is set to the correct ARC length wich is supported by the RC. 
  LengthACR                 : UINT := 50;  
  /// Highest index of available tools on the RC.
  HighestToolIndex          : USINT;
  /// Highest index of available frames on the RC.
  HighestFrameIndex         : USINT;
  /// Highest index of available loads on the RC.
  HighestLoadIndex          : USINT;
  /// Highest index of available work areas on the RC.
  HighestWorkAreaIndex      : USINT;
  /// Datas which are synchronized
  DataInSync                : DataInSync;
  /// Index of tool changed on RC
  ChangeIndexTool           : USINT;
  /// Index of frame changed on RC
  ChangeIndexFrame          : USINT;
  /// Index of load changed on RC
  ChangeIndexLoad           : USINT;
  ///Index of work area changed on RC
  ChangeIndexWorkArea       : USINT;
  /// Working hours of an RA connected to the RC
  RAWorkingHours            : UDINT;
  /// Signals that a brake test is required in the defined monitoring time (see chapter 6.5.27)
  BrakeTestRequired         : BOOL;
  /// StepMode is active and set to ExactStop (see chapter 6.1.3)
  StepModeExactStopActive   : BOOL;
  /// StepMode is active and set to Blending (see chapter 6.1.3)
  StepModeBlendingActive    : BOOL;
  /// PathAccuracyMode is active (see chapter 6.5.22)
  PathAccuracyMode          : BOOL;
  /// AvoidSingularity is active (see chapter 6.5.23)
  AvoidSingularity          : BOOL;
  /// CollisionDetection is active (see chapter 6.5.35)
  CollisionDetectionEnabled : BOOL;
  /// Cyclic dynamics status bit Accelerating is supported by RC (see chapter 5.5.3.2)
  AcceleratingSupported     : BOOL;
  /// Cyclic dynamics status bit Decelerating is supported by RC (see chapter 5.5.3.2)
  DecceleratingSupported    : BOOL;
  /// Cyclic dynamics status bit ConstantVelocity is supported by RC (see chapter 5.5.3.2)
  ConstantVelocitySupported : BOOL;
  /// Total system hours of an RA connected to the RC. Must not be modifiable by the user.
  /// •  0: Invalid
  /// • >1: Total system hours
  RCWorkingHours            : UDINT;
END_STRUCT
END_TYPE

// Library/Structures/AxesGroup/Parameter/AxesGroupParameter
{attribute 'pack_mode' := '1'} 
// ------------------------------------------------------------------------- 
//  SRCI Robot Library                                                
// ------------------------------------------------------------------------- 
//                                                                           
//  Object:      AxesGroupParameter                                       
//  Author:      Thorsten Brach                                                
//  Date:        2024-06-01
//
//  Description:                                              
//   
//                                                                           
//  Copyright: 
//    (C) 2024 Thorsten Brach. All rights reserved                                                                                                                                            
//             Licensed under the LGPL-3.0 license.
//                                                                           
//  Disclaimer:                                                                           
//    This project is provided without any guarantee and can be used for   
//    private and commercial purposes. Any use is at the user’s 
//    own risk and responsibility.
//
// -------------------------------------------------------------------------
TYPE AxesGroupParameter :
STRUCT
  /// PLC specific data
  Plc            : AxesGroupParameterPlc;
  /// RC data read by the function "ReadRobotData" (see chapter 6.1.2)
  Rob            : AxesGroupParameterRob;

(*  /// Optional cyclic data configuration
  OptionalCyclic : AxesGroupParameterOptionalCyclic;
*)  
END_STRUCT
END_TYPE

// Library/Structures/AxesGroup/State/DataChanged/AxesGroupStateDataChanged
{attribute 'pack_mode' := '1'} 
// ------------------------------------------------------------------------- 
//  SRCI Robot Library                                                
// ------------------------------------------------------------------------- 
//                                                                           
//  Object:      AxesGroupStateDataChanged                                       
//  Author:      Thorsten Brach                                                
//  Date:        2024-06-01
//
//  Description:                                              
//   
//                                                                           
//  Copyright: 
//    (C) 2024 Thorsten Brach. All rights reserved                                                                                                                                            
//             Licensed under the LGPL-3.0 license.
//                                                                           
//  Disclaimer:                                                                           
//    This project is provided without any guarantee and can be used for   
//    private and commercial purposes. Any use is at the user’s 
//    own risk and responsibility.
//
// -------------------------------------------------------------------------
TYPE AxesGroupStateDataChanged :
STRUCT
  /// indicates that tool data has changed
  Tool             : ARRAY[0..255] OF BOOL;
  /// indicates that frame data has changed
  Frame            : ARRAY[0..255] OF BOOL;
  /// indicates that load data has changed
  Load             : ARRAY[0..255] OF BOOL;
  /// indicates that work area has changed
  WorkArea         : ARRAY[0..255] OF BOOL;
  /// indicates that default dynamic has changed
  DefaultDynamic   : BOOL;
  /// indicates that reference dynamic has changed
  ReferenceDynamic : BOOL;
  /// indicates that software limits has changed
  SwLimits         : BOOL;
END_STRUCT
END_TYPE

// Library/Structures/AxesGroup/State/ResetMsg/AxesGroupStateResetMsg
{attribute 'pack_mode' := '1'} 
// ------------------------------------------------------------------------- 
//  SRCI Robot Library                                                
// ------------------------------------------------------------------------- 
//                                                                           
//  Object:      AxesGroupStateResetMsg                                       
//  Author:      Thorsten Brach                                                
//  Date:        2024-06-01
//
//  Description:                                              
//   
//                                                                           
//  Copyright: 
//    (C) 2024 Thorsten Brach. All rights reserved                                                                                                                                            
//             Licensed under the LGPL-3.0 license.
//                                                                           
//  Disclaimer:                                                                           
//    This project is provided without any guarantee and can be used for   
//    private and commercial purposes. Any use is at the user’s 
//    own risk and responsibility.
//
// -------------------------------------------------------------------------
TYPE AxesGroupStateResetMsg :
STRUCT
  ///
  Reset     : BOOL;
  ///
  ResetTime : DT;
END_STRUCT
END_TYPE

// Library/Structures/AxesGroup/State/RobotData/AxesGroupRobotData
{attribute 'pack_mode' := '1'} 
// ------------------------------------------------------------------------- 
//  SRCI Robot Library                                                
// ------------------------------------------------------------------------- 
//                                                                           
//  Object:      AxesGroupRobotData                                       
//  Author:      Thorsten Brach                                                
//  Date:        2024-11-29
//
//  Description:                                              
//   
//                                                                           
//  Copyright: 
//    (C) 2024 Thorsten Brach. All rights reserved                                                                                                                                            
//             Licensed under the LGPL-3.0 license.
//                                                                           
//  Disclaimer:                                                                           
//    This project is provided without any guarantee and can be used for   
//    private and commercial purposes. Any use is at the user’s 
//    own risk and responsibility.
//
// -------------------------------------------------------------------------
TYPE AxesGroupRobotData EXTENDS ReadRobotDataOutCmd :
STRUCT
  dummy : bool;
END_STRUCT
END_TYPE

// Library/Structures/AxesGroup/State/Synchronizing/AxesGroupStateSynchronizing
{attribute 'pack_mode' := '1'} 
// ------------------------------------------------------------------------- 
//  SRCI Robot Library                                                
// ------------------------------------------------------------------------- 
//                                                                           
//  Object:      AxesGroupStateSynchronizing                                       
//  Author:      Thorsten Brach                                                
//  Date:        2024-06-01
//
//  Description:                                              
//   
//                                                                           
//  Copyright: 
//    (C) 2024 Thorsten Brach. All rights reserved                                                                                                                                            
//             Licensed under the LGPL-3.0 license.
//                                                                           
//  Disclaimer:                                                                           
//    This project is provided without any guarantee and can be used for   
//    private and commercial purposes. Any use is at the user’s 
//    own risk and responsibility.
//
// -------------------------------------------------------------------------
TYPE AxesGroupStateSynchronizing :
STRUCT
  /// indicates that the tooldata are synchronized
  Tool           : BOOL;
  /// indicates that the framedata are synchronized
  Frame          : BOOL;
  /// indicates that the loaddata are synchronized
  Load           : BOOL;
  /// indicates that the work areas are synchronized
  WorkAreas      : BOOL;
  /// indicates that the reference-dynamics are synchronized
  RefDynamic     : BOOL;
  /// indicates that the default-dynamics are synchronized
  DefaultDynamic : BOOL;
  /// indicates that the software limits are synchronized
  SwLimits       : BOOL;
END_STRUCT
END_TYPE

// Library/Structures/AxesGroup/State/SyncState/AxesGroupStateSyncState
{attribute 'pack_mode' := '1'} 
// ------------------------------------------------------------------------- 
//  SRCI Robot Library                                                
// ------------------------------------------------------------------------- 
//                                                                           
//  Object:      AxesGroupStateSyncState                                       
//  Author:      Thorsten Brach                                                
//  Date:        2024-06-01
//
//  Description:                                              
//   
//                                                                           
//  Copyright: 
//    (C) 2024 Thorsten Brach. All rights reserved                                                                                                                                            
//             Licensed under the LGPL-3.0 license.
//                                                                           
//  Disclaimer:                                                                           
//    This project is provided without any guarantee and can be used for   
//    private and commercial purposes. Any use is at the user’s 
//    own risk and responsibility.
//
// -------------------------------------------------------------------------
TYPE AxesGroupStateSyncState :
STRUCT
  /// Bit 00: Tool
  Tool             : BOOL;
  /// Bit 01: Frame
  Frame            : BOOL;
  /// Bit 02: Load
  Load             : BOOL;
  /// Bit 03: WorkArea
  WorkArea         : BOOL;
  /// Bit 04: SwLimits
  SwLimits         : BOOL;
  /// Bit 05: DefaultDynamic
  DefaultDynamic   : BOOL;
  /// Bit 06: ReferenceDynamic
  ReferenceDynamic : BOOL;
  /// Bit 07:
  Bit07            : BOOL;
  /// Bit 08:
  Bit08            : BOOL;
  /// Bit 09:
  Bit09            : BOOL;
  /// Bit 10:
  Bit10            : BOOL;
  /// Bit 11:
  Bit11            : BOOL;
  /// Bit 12:
  Bit12            : BOOL;
  /// Bit 13:
  Bit13            : BOOL;
  /// Bit 14:
  Bit14            : BOOL;
  /// Bit 15:
  Bit15            : BOOL;  
END_STRUCT
END_TYPE

// Library/Structures/AxesGroup/State/SyncState/AxesGroupStateSyncStateNo
{attribute 'pack_mode' := '1'} 
// ------------------------------------------------------------------------- 
//  SRCI Robot Library                                                
// ------------------------------------------------------------------------- 
//                                                                           
//  Object:      AxesGroupStateSyncStateNo                                       
//  Author:      Thorsten Brach                                                
//  Date:        2024-06-01
//
//  Description:                                              
//   
//                                                                           
//  Copyright: 
//    (C) 2024 Thorsten Brach. All rights reserved                                                                                                                                            
//             Licensed under the LGPL-3.0 license.
//                                                                           
//  Disclaimer:                                                                           
//    This project is provided without any guarantee and can be used for   
//    private and commercial purposes. Any use is at the user’s 
//    own risk and responsibility.
//
// -------------------------------------------------------------------------
TYPE AxesGroupStateSyncStateNo :
STRUCT
  /// Ammount of unsynchronized tool data
  Tool     : USINT;
  /// Ammount of unsynchronized frame data
  Frame    : USINT;
  /// Ammount of unsynchronized load data
  Load     : USINT;
  /// Ammount of unsynchronized word areas
  WorkArea : USINT;    
END_STRUCT
END_TYPE

// Library/Structures/AxesGroup/State/SyncState/AxesGroupStateSyncStatePlc
{attribute 'pack_mode' := '1'} 
// ------------------------------------------------------------------------- 
//  SRCI Robot Library                                                
// ------------------------------------------------------------------------- 
//                                                                           
//  Object:      AxesGroupStateSyncStatePlc                                       
//  Author:      Thorsten Brach                                                
//  Date:        2024-06-01
//
//  Description:                                              
//   
//                                                                           
//  Copyright: 
//    (C) 2024 Thorsten Brach. All rights reserved                                                                                                                                            
//             Licensed under the LGPL-3.0 license.
//                                                                           
//  Disclaimer:                                                                           
//    This project is provided without any guarantee and can be used for   
//    private and commercial purposes. Any use is at the user’s 
//    own risk and responsibility.
//
// -------------------------------------------------------------------------
TYPE AxesGroupStateSyncStatePlc :
STRUCT
  ///
  InSync   : AxesGroupStateSyncState;
END_STRUCT
END_TYPE

// Library/Structures/AxesGroup/State/SyncState/AxesGroupStateSyncStateRob
{attribute 'pack_mode' := '1'} 
// ------------------------------------------------------------------------- 
//  SRCI Robot Library                                                
// ------------------------------------------------------------------------- 
//                                                                           
//  Object:      AxesGroupStateSyncStateRob                                       
//  Author:      Thorsten Brach                                                
//  Date:        2024-06-01
//
//  Description:                                              
//   
//                                                                           
//  Copyright: 
//    (C) 2024 Thorsten Brach. All rights reserved                                                                                                                                            
//             Licensed under the LGPL-3.0 license.
//                                                                           
//  Disclaimer:                                                                           
//    This project is provided without any guarantee and can be used for   
//    private and commercial purposes. Any use is at the user’s 
//    own risk and responsibility.
//
// -------------------------------------------------------------------------
TYPE AxesGroupStateSyncStateRob :
STRUCT
  ///
  InSync   : AxesGroupStateSyncState;
  ///
  UnSyncNo : AxesGroupStateSyncStateNo;
END_STRUCT
END_TYPE

// Library/Structures/AxesGroup/State/AxesGroupState
{attribute 'pack_mode' := '1'} 
// ------------------------------------------------------------------------- 
//  SRCI Robot Library                                                
// ------------------------------------------------------------------------- 
//                                                                           
//  Object:      AxesGroupState                                       
//  Author:      Thorsten Brach                                                
//  Date:        2024-06-01
//
//  Description:                                              
//   
//                                                                           
//  Copyright: 
//    (C) 2024 Thorsten Brach. All rights reserved                                                                                                                                            
//             Licensed under the LGPL-3.0 license.
//                                                                           
//  Disclaimer:                                                                           
//    This project is provided without any guarantee and can be used for   
//    private and commercial purposes. Any use is at the user’s 
//    own risk and responsibility.
//
// -------------------------------------------------------------------------
TYPE AxesGroupState :
STRUCT
  ///
  FatalErrorClient  : BOOL;
  ///
  Initialized       : BOOL;
  ///
  Synchronized      : BOOL;
  ///
  Synchronizing     : AxesGroupStateSynchronizing;
  ///
  AliveOk           : BOOL;
  ///
  CMDsEnabled       : BOOL;
  ///
  ConfigExchanged   : BOOL;
  /// 
  RobotIdent        : DT;
  ///
  DataChanged       : AxesGroupStateDataChanged;
  ///
  SyncStatePlc      : AxesGroupStateSyncStatePlc;
  /// 
  SyncStateRc       : AxesGroupStateSyncStateRob;
  ///
  ResetMsg          : AxesGroupStateResetMsg;
  ///
  IncrementFastStop : BOOL;
  /// Robot Data
  RobotData         : AxesGroupRobotData;
END_STRUCT
END_TYPE

// Library/Structures/AxesGroup/AxesGroup
{attribute 'pack_mode' := '1'} 
// ------------------------------------------------------------------------- 
//  SRCI Robot Library                                                
// ------------------------------------------------------------------------- 
//                                                                           
//  Object:      AxesGroup                                       
//  Author:      Thorsten Brach                                                
//  Date:        2024-06-01
//
//  Description:                                              
//   
//                                                                           
//  Copyright: 
//    (C) 2024 Thorsten Brach. All rights reserved                                                                                                                                            
//             Licensed under the LGPL-3.0 license.
//                                                                           
//  Disclaimer:                                                                           
//    This project is provided without any guarantee and can be used for   
//    private and commercial purposes. Any use is at the user’s 
//    own risk and responsibility.
//
// -------------------------------------------------------------------------
TYPE AxesGroup :
STRUCT
  /// Parameter 
  Parameter      : AxesGroupParameter;
  /// RI state information (see chapter 5.5.3) 
  State          : AxesGroupState;
  /// RC, RA, RI, and CMD warnings and errors (see chapter 5.5.11)
  MessageLog     : AxesGroupMessageLogFB;
  /// Cyclic data exchanged between server and client (see chapter 5.6.6.5) 
  Cyclic         : AxesGroupCyclic;
  /// Optional cyclic data exchanged between server and client (see chapter 5.6.6.2)
  CyclicOptional : AxesGroupCyclicOptionalData;
  /// Execution order list and ACR entries (see chapter 5.6.4.2) 
  Acyclic        : AxesGroupAcyclic;
  /// Internal data
  InternalData   : AxesGroupInternalData;
END_STRUCT
END_TYPE

// Library/Structures/Cartesian/RobotCartesianForce
{attribute 'pack_mode' := '1'} 
// ------------------------------------------------------------------------- 
//  SRCI Robot Library                                                
// ------------------------------------------------------------------------- 
//                                                                           
//  Object:      RobotCartesianForce                                       
//  Author:      Thorsten Brach                                                
//  Date:        2024-06-01
//
//  Description:                                              
//   
//                                                                           
//  Copyright: 
//    (C) 2024 Thorsten Brach. All rights reserved                                                                                                                                            
//             Licensed under the LGPL-3.0 license.
//                                                                           
//  Disclaimer:                                                                           
//    This project is provided without any guarantee and can be used for   
//    private and commercial purposes. Any use is at the user’s 
//    own risk and responsibility.
//
// -------------------------------------------------------------------------
TYPE RobotCartesianForce :
STRUCT
  /// Force on the X-Axis
  X : REAL;
  /// Force on the Y-Axis
  Y : REAL;
  /// Force on the Z-Axis
  Z : REAL;
  /// Force around the X-Axis (RX)
  Rx : REAL;
  /// Force around the Y-Axis (RY)
  Ry : REAL;
  /// Force around the Z-Axis (RZ)
  Rz : REAL;
  /// Force of first external axis
  E1 : REAL;
  /// Force of second external axis
  E2 : REAL;
  /// Force of third external axis
  E3 : REAL;
  /// Force of fourth external axis
  E4 : REAL;
  /// Force of fifth external axis
  E5 : REAL;
  /// Force of sixth external axis
  E6 : REAL;    
END_STRUCT
END_TYPE

// Library/Structures/Cartesian/RobotCartesianForceExt
{attribute 'pack_mode' := '1'} 
// ------------------------------------------------------------------------- 
//  SRCI Robot Library                                                
// ------------------------------------------------------------------------- 
//                                                                           
//  Object:      RobotCartesianForceExt                                       
//  Author:      Thorsten Brach                                                
//  Date:        2024-06-01
//
//  Description:                                              
//   
//                                                                           
//  Copyright: 
//    (C) 2024 Thorsten Brach. All rights reserved                                                                                                                                            
//             Licensed under the LGPL-3.0 license.
//                                                                           
//  Disclaimer:                                                                           
//    This project is provided without any guarantee and can be used for   
//    private and commercial purposes. Any use is at the user’s 
//    own risk and responsibility.
//
// -------------------------------------------------------------------------
TYPE RobotCartesianForceExt :
STRUCT
  /// Force on the first external axis
  E1 : REAL;
  /// Force of second external axis
  E2 : REAL;
  /// Force of third external axis
  E3 : REAL;
  /// Force of fourth external axis
  E4 : REAL;
  /// Force of fifth external axis
  E5 : REAL;
  /// Force of sixth external axis
  E6 : REAL;  
END_STRUCT
END_TYPE

// Library/Structures/Cartesian/RobotCartesianForceShort
{attribute 'pack_mode' := '1'} 
// ------------------------------------------------------------------------- 
//  SRCI Robot Library                                                
// ------------------------------------------------------------------------- 
//                                                                           
//  Object:      RobotCartesianForceShort                                       
//  Author:      Thorsten Brach                                                
//  Date:        2024-06-01
//
//  Description:                                              
//   
//                                                                           
//  Copyright: 
//    (C) 2024 Thorsten Brach. All rights reserved                                                                                                                                            
//             Licensed under the LGPL-3.0 license.
//                                                                           
//  Disclaimer:                                                                           
//    This project is provided without any guarantee and can be used for   
//    private and commercial purposes. Any use is at the user’s 
//    own risk and responsibility.
//
// -------------------------------------------------------------------------
TYPE RobotCartesianForceShort :
STRUCT
  /// Force on the X-Axis
  X : REAL;
  /// Force on the Y-Axis
  Y : REAL;
  /// Force on the Z-Axis
  Z : REAL;
  /// Force around the X-Axis (RX)
  Rx : REAL;
  /// Force around the Y-Axis (RY)
  Ry : REAL;
  /// Force around the Z-Axis (RZ)
  Rz : REAL;
END_STRUCT
END_TYPE

